Yaskawa INFORM job: OPEN-CURTAIN.JBI

/JOB
//NAME OPEN-CURTAIN
//POS
///NPOS 0,0,0,0,0,0
//INST
///DATE 2018/09/03 10:50
///ATTR SC,RW
NOP
DOUT OT#(15) OFF
TIMER T=0.20
DOUT OT#(5) ON
WAIT IN#(15)=ON T=20.00
*error
IFTHEN IN#(15)=OFF
	 SETUALM 8000 "Curtain is not open" 0
	 PAUSE
	 JUMP *error
ENDIF
DOUT OT#(5) OFF
DOUT OT#(15) OFF
INC B007
*END
END
